Yaskawa INFORM job: SIDEB-30.JBI

/JOB
//NAME SIDEB-30
///FOLDERNAME MASTER
//POS
///NPOS 0,0,1,0,0,0
///TOOL 0
///POSTYPE PULSE
///PULSE
EC00000=-101065
//INST
///DATE 2021/10/29 11:49
///ATTR SC,RO
///GROUP1 ST3
NOP
MOVJ EC00000 VJ=50.00
END
